PROGRAM MAIN
VAR
	NCI : NCICHannel;
END_VAR

END_PROGRAM

(* stored: Version 1.1.0.1, ProductVersion 3.1.4018.5
   POU MAIN: Id {85512ce5-5fef-4ca9-8013-0a3b70b6fd2d}, SpecialFunc None *)
